       // Index 1
       IF "HMI_Interface_Overview".homeCodition[7].pageIndex = 1 THEN
           "HMI_Interface_Overview".homeCodition[7].emOverviewTitle := WSTRING#'Home Condition 1';
           "HMI_Interface_Overview".homeCodition[7].emOverviewCmName[0] := WSTRING#'Hot Press Right Servo Press';
           "HMI_Interface_Overview".homeCodition[7].emOverviewCmName[1] := WSTRING#'Hot Press Right Stage Lift Front';
           "HMI_Interface_Overview".homeCodition[7].emOverviewCmName[2] := WSTRING#'Hot Press Right Stage Lift Rear';
           "HMI_Interface_Overview".homeCodition[7].emOverviewCmName[3] := WSTRING#'Hot Press Right JR Detect';
           "HMI_Interface_Overview".homeCodition[7].emOverviewCmName[4] := WSTRING#'Spare';
           "HMI_Interface_Overview".homeCodition[7].emOverviewCmName[5] := WSTRING#'Spare';
           "HMI_Interface_Overview".homeCodition[7].emOverviewCmName[6] := WSTRING#'Spare';
           "HMI_Interface_Overview".homeCodition[7].emOverviewCmName[7] := WSTRING#'Spare';
           "HMI_Interface_Overview".homeCodition[7].emOverviewCmName[8] := WSTRING#'Spare';
           "HMI_Interface_Overview".homeCodition[7].emOverviewCmName[9] := WSTRING#'Spare';
           "HMI_Interface_Overview".homeCodition[7].emOverviewCmName[10] := WSTRING#'Spare';
           "HMI_Interface_Overview".homeCodition[7].emOverviewCmName[11] := WSTRING#'Spare';
           "HMI_Interface_Overview".homeCodition[7].emOverviewCmName[12] := WSTRING#'Spare';
           "HMI_Interface_Overview".homeCodition[7].emOverviewCmName[13] := WSTRING#'Spare';
           "HMI_Interface_Overview".homeCodition[7].emOverviewCmPositionName[0] := WSTRING#'Home Position';
           "HMI_Interface_Overview".homeCodition[7].emOverviewCmPositionName[1] := WSTRING#'Down';
           "HMI_Interface_Overview".homeCodition[7].emOverviewCmPositionName[2] := WSTRING#'Down';
           "HMI_Interface_Overview".homeCodition[7].emOverviewCmPositionName[3] := WSTRING#'Detect';
           "HMI_Interface_Overview".homeCodition[7].emOverviewCmPositionName[4] := WSTRING#'Spare';
           "HMI_Interface_Overview".homeCodition[7].emOverviewCmPositionName[5] := WSTRING#'Spare';
           "HMI_Interface_Overview".homeCodition[7].emOverviewCmPositionName[6] := WSTRING#'Spare';
           "HMI_Interface_Overview".homeCodition[7].emOverviewCmPositionName[7] := WSTRING#'Spare';
           "HMI_Interface_Overview".homeCodition[7].emOverviewCmPositionName[8] := WSTRING#'Spare';
           "HMI_Interface_Overview".homeCodition[7].emOverviewCmPositionName[9] := WSTRING#'Spare';
           "HMI_Interface_Overview".homeCodition[7].emOverviewCmPositionName[10] := WSTRING#'Spare';
           "HMI_Interface_Overview".homeCodition[7].emOverviewCmPositionName[11] := WSTRING#'Spare';
           "HMI_Interface_Overview".homeCodition[7].emOverviewCmPositionName[12] := WSTRING#'Spare';
           "HMI_Interface_Overview".homeCodition[7].emOverviewCmPositionName[13] := WSTRING#'Spare';
           IF NOT #statLampControl THEN
               "HMI_Interface_Overview".homeCodition[7].emOverviewHomeLampOn[0] := "Unit1.Em7.HmiInterface".cmHotPressRightServoPress.monitoring.profinetInput."HOME-POS-REACHED";
               "HMI_Interface_Overview".homeCodition[7].emOverviewHomeLampOn[1] := "Unit1.Em7.HmiInterface".cmHotPressRightStageLiftFrontUpDown.monitoring.inWorkPos;
               "HMI_Interface_Overview".homeCodition[7].emOverviewHomeLampOn[2] := "Unit1.Em7.HmiInterface".cmHotPressRightStageLiftRearUpDown.monitoring.inWorkPos;
               "HMI_Interface_Overview".homeCodition[7].emOverviewHomeLampOn[3] := "Unit1.Em7.HmiInterface".cmHotPressRightJRDetect.monitoring.processValue;
               "HMI_Interface_Overview".homeCodition[7].emOverviewHomeLampOn[4] := FALSE;
               "HMI_Interface_Overview".homeCodition[7].emOverviewHomeLampOn[5] := FALSE;
               "HMI_Interface_Overview".homeCodition[7].emOverviewHomeLampOn[6] := FALSE;
               "HMI_Interface_Overview".homeCodition[7].emOverviewHomeLampOn[7] := FALSE;
               "HMI_Interface_Overview".homeCodition[7].emOverviewHomeLampOn[8] := FALSE;
               "HMI_Interface_Overview".homeCodition[7].emOverviewHomeLampOn[9] := FALSE;
               "HMI_Interface_Overview".homeCodition[7].emOverviewHomeLampOn[10] := FALSE;
               "HMI_Interface_Overview".homeCodition[7].emOverviewHomeLampOn[11] := FALSE;
               "HMI_Interface_Overview".homeCodition[7].emOverviewHomeLampOn[12] := FALSE;
               "HMI_Interface_Overview".homeCodition[7].emOverviewHomeLampOn[13] := FALSE;
           END_IF;
       END_IF;

   END_REGION
END_REGION

REGION Network 38 (SCL): Em 8 Page Index Mapping
   REGION Page Index

       // Index 0
       IF "HMI_Interface_Overview".homeCodition[8].pageIndex = 0 THEN
           "HMI_Interface_Overview".homeCodition[8].emOverviewTitle := WSTRING#'Home Condition 0';
           "HMI_Interface_Overview".homeCodition[8].emOverviewCmName[0] := WSTRING#'Thickness Z-Axis';
           "HMI_Interface_Overview".homeCodition[8].emOverviewCmName[1] := WSTRING#'Hipot & Thickness Servo Press';
           "HMI_Interface_Overview".homeCodition[8].emOverviewCmName[2] := WSTRING#'Hipot Tab Contactor Left';
           "HMI_Interface_Overview".homeCodition[8].emOverviewCmName[3] := WSTRING#'Hipot Tab Contactor Right';
           "HMI_Interface_Overview".homeCodition[8].emOverviewCmName[4] := WSTRING#'Hipot Tab Contactor';
           "HMI_Interface_Overview".homeCodition[8].emOverviewCmName[5] := WSTRING#'Hipot & Thickness Stage Lift Front';
           "HMI_Interface_Overview".homeCodition[8].emOverviewCmName[6] := WSTRING#'Hipot & Thickness Stage Lift Rear';
           "HMI_Interface_Overview".homeCodition[8].emOverviewCmName[7] := WSTRING#'Hipot & Thickness JR Detect';
           "HMI_Interface_Overview".homeCodition[8].emOverviewCmName[8] := WSTRING#'Spare';
           "HMI_Interface_Overview".homeCodition[8].emOverviewCmName[9] := WSTRING#'Spare';
           "HMI_Interface_Overview".homeCodition[8].emOverviewCmName[10] := WSTRING#'Spare';
           "HMI_Interface_Overview".homeCodition[8].emOverviewCmName[11] := WSTRING#'Spare';
           "HMI_Interface_Overview".homeCodition[8].emOverviewCmName[12] := WSTRING#'Spare';
           "HMI_Interface_Overview".homeCodition[8].emOverviewCmName[13] := WSTRING#'Spare';
           "HMI_Interface_Overview".homeCodition[8].emOverviewCmPositionName[0] := WSTRING#'Wait Position';
           "HMI_Interface_Overview".homeCodition[8].emOverviewCmPositionName[1] := WSTRING#'Home Position';
           "HMI_Interface_Overview".homeCodition[8].emOverviewCmPositionName[2] := WSTRING#'Open';
           "HMI_Interface_Overview".homeCodition[8].emOverviewCmPositionName[3] := WSTRING#'Open';
           "HMI_Interface_Overview".homeCodition[8].emOverviewCmPositionName[4] := WSTRING#'Backward';
           "HMI_Interface_Overview".homeCodition[8].emOverviewCmPositionName[5] := WSTRING#'Down';
           "HMI_Interface_Overview".homeCodition[8].emOverviewCmPositionName[6] := WSTRING#'Down';
           "HMI_Interface_Overview".homeCodition[8].emOverviewCmPositionName[7] := WSTRING#'Not Detect';
           "HMI_Interface_Overview".homeCodition[8].emOverviewCmPositionName[8] := WSTRING#'Spare';
           "HMI_Interface_Overview".homeCodition[8].emOverviewCmPositionName[9] := WSTRING#'Spare';
           "HMI_Interface_Overview".homeCodition[8].emOverviewCmPositionName[10] := WSTRING#'Spare';
           "HMI_Interface_Overview".homeCodition[8].emOverviewCmPositionName[11] := WSTRING#'Spare';
           "HMI_Interface_Overview".homeCodition[8].emOverviewCmPositionName[12] := WSTRING#'Spare';
           "HMI_Interface_Overview".homeCodition[8].emOverviewCmPositionName[13] := WSTRING#'Spare';
           IF NOT #statLampControl THEN
               "HMI_Interface_Overview".homeCodition[8].emOverviewHomeLampOn[0] := "Unit1.Em8.HmiInterface".cm.softcam.thicknessAxisZ.pos00_wait.inPos;
               "HMI_Interface_Overview".homeCodition[8].emOverviewHomeLampOn[1] := "Unit1.Em8.HmiInterface".cmHipotThicknessServoPress.monitoring.profinetInput."HOME-POS-REACHED";
               "HMI_Interface_Overview".homeCodition[8].emOverviewHomeLampOn[2] := "Unit1.Em8.HmiInterface".cmHipotTabContactorLeftOpenClose.monitoring.inHomePos;
               "HMI_Interface_Overview".homeCodition[8].emOverviewHomeLampOn[3] := "Unit1.Em8.HmiInterface".cmHipotTabContactorRightOpenClose.monitoring.inHomePos;
               "HMI_Interface_Overview".homeCodition[8].emOverviewHomeLampOn[4] := "Unit1.Em8.HmiInterface".cmHipotTabContactorBwdFwd.monitoring.inHomePos;
               "HMI_Interface_Overview".homeCodition[8].emOverviewHomeLampOn[5] := "Unit1.Em8.HmiInterface".cmHipotThicknessStageLiftFrontUpDown.monitoring.inWorkPos;
               "HMI_Interface_Overview".homeCodition[8].emOverviewHomeLampOn[6] := "Unit1.Em8.HmiInterface".cmHipotThicknessStageLiftRearUpDown.monitoring.inWorkPos;
               "HMI_Interface_Overview".homeCodition[8].emOverviewHomeLampOn[7] := NOT "Unit1.Em8.HmiInterface".cmHipotThicknessJRDetect.monitoring.processValue;
               "HMI_Interface_Overview".homeCodition[8].emOverviewHomeLampOn[8] := FALSE;
               "HMI_Interface_Overview".homeCodition[8].emOverviewHomeLampOn[9] := FALSE;
               "HMI_Interface_Overview".homeCodition[8].emOverviewHomeLampOn[10] := FALSE;
               "HMI_Interface_Overview".homeCodition[8].emOverviewHomeLampOn[11] := FALSE;
               "HMI_Interface_Overview".homeCodition[8].emOverviewHomeLampOn[12] := FALSE;
               "HMI_Interface_Overview".homeCodition[8].emOverviewHomeLampOn[13] := FALSE;
           END_IF;
       END_IF;

       // Index 1
       IF "HMI_Interface_Overview".homeCodition[8].pageIndex = 1 THEN
           "HMI_Interface_Overview".homeCodition[8].emOverviewTitle := WSTRING#'Home Condition 1';
           "HMI_Interface_Overview".homeCodition[8].emOverviewCmName[0] := WSTRING#'Thickness Z-Axis';
           "HMI_Interface_Overview".homeCodition[8].emOverviewCmName[1] := WSTRING#'Hipot & Thickness Servo Press';
           "HMI_Interface_Overview".homeCodition[8].emOverviewCmName[2] := WSTRING#'Hipot Tab Contactor Left';
           "HMI_Interface_Overview".homeCodition[8].emOverviewCmName[3] := WSTRING#'Hipot Tab Contactor Right';
           "HMI_Interface_Overview".homeCodition[8].emOverviewCmName[4] := WSTRING#'Hipot Tab Contactor';
           "HMI_Interface_Overview".homeCodition[8].emOverviewCmName[5] := WSTRING#'Hipot & Thickness Stage Lift Front';
           "HMI_Interface_Overview".homeCodition[8].emOverviewCmName[6] := WSTRING#'Hipot & Thickness Stage Lift Rear';
           "HMI_Interface_Overview".homeCodition[8].emOverviewCmName[7] := WSTRING#'Hipot & Thickness JR Detect';
           "HMI_Interface_Overview".homeCodition[8].emOverviewCmName[8] := WSTRING#'Spare';
           "HMI_Interface_Overview".homeCodition[8].emOverviewCmName[9] := WSTRING#'Spare';
           "HMI_Interface_Overview".homeCodition[8].emOverviewCmName[10] := WSTRING#'Spare';
           "HMI_Interface_Overview".homeCodition[8].emOverviewCmName[11] := WSTRING#'Spare';
           "HMI_Interface_Overview".homeCodition[8].emOverviewCmName[12] := WSTRING#'Spare';
           "HMI_Interface_Overview".homeCodition[8].emOverviewCmName[13] := WSTRING#'Spare';
           "HMI_Interface_Overview".homeCodition[8].emOverviewCmPositionName[0] := WSTRING#'Wait Position';
           "HMI_Interface_Overview".homeCodition[8].emOverviewCmPositionName[1] := WSTRING#'Home Position';
           "HMI_Interface_Overview".homeCodition[8].emOverviewCmPositionName[2] := WSTRING#'Open';
           "HMI_Interface_Overview".homeCodition[8].emOverviewCmPositionName[3] := WSTRING#'Open';
           "HMI_Interface_Overview".homeCodition[8].emOverviewCmPositionName[4] := WSTRING#'Backward';
           "HMI_Interface_Overview".homeCodition[8].emOverviewCmPositionName[5] := WSTRING#'Down';
           "HMI_Interface_Overview".homeCodition[8].emOverviewCmPositionName[6] := WSTRING#'Down';
           "HMI_Interface_Overview".homeCodition[8].emOverviewCmPositionName[7] := WSTRING#'Detect';
           "HMI_Interface_Overview".homeCodition[8].emOverviewCmPositionName[8] := WSTRING#'Spare';
           "HMI_Interface_Overview".homeCodition[8].emOverviewCmPositionName[9] := WSTRING#'Spare';
           "HMI_Interface_Overview".homeCodition[8].emOverviewCmPositionName[10] := WSTRING#'Spare';
           "HMI_Interface_Overview".homeCodition[8].emOverviewCmPositionName[11] := WSTRING#'Spare';
           "HMI_Interface_Overview".homeCodition[8].emOverviewCmPositionName[12] := WSTRING#'Spare';
           "HMI_Interface_Overview".homeCodition[8].emOverviewCmPositionName[13] := WSTRING#'Spare';
           IF NOT #statLampControl THEN
               "HMI_Interface_Overview".homeCodition[8].emOverviewHomeLampOn[0] := "Unit1.Em8.HmiInterface".cm.softcam.thicknessAxisZ.pos00_wait.inPos;
               "HMI_Interface_Overview".homeCodition[8].emOverviewHomeLampOn[1] := "Unit1.Em8.HmiInterface".cmHipotThicknessServoPress.monitoring.profinetInput."HOME-POS-REACHED";
               "HMI_Interface_Overview".homeCodition[8].emOverviewHomeLampOn[2] := "Unit1.Em8.HmiInterface".cmHipotTabContactorLeftOpenClose.monitoring.inHomePos;
               "HMI_Interface_Overview".homeCodition[8].emOverviewHomeLampOn[3] := "Unit1.Em8.HmiInterface".cmHipotTabContactorRightOpenClose.monitoring.inHomePos;
               "HMI_Interface_Overview".homeCodition[8].emOverviewHomeLampOn[4] := "Unit1.Em8.HmiInterface".cmHipotTabContactorBwdFwd.monitoring.inHomePos;
               "HMI_Interface_Overview".homeCodition[8].emOverviewHomeLampOn[5] := "Unit1.Em8.HmiInterface".cmHipotThicknessStageLiftFrontUpDown.monitoring.inWorkPos;
               "HMI_Interface_Overview".homeCodition[8].emOverviewHomeLampOn[6] := "Unit1.Em8.HmiInterface".cmHipotThicknessStageLiftRearUpDown.monitoring.inWorkPos;
               "HMI_Interface_Overview".homeCodition[8].emOverviewHomeLampOn[7] := "Unit1.Em8.HmiInterface".cmHipotThicknessJRDetect.monitoring.processValue;
               "HMI_Interface_Overview".homeCodition[8].emOverviewHomeLampOn[8] := FALSE;
               "HMI_Interface_Overview".homeCodition[8].emOverviewHomeLampOn[9] := FALSE;
               "HMI_Interface_Overview".homeCodition[8].emOverviewHomeLampOn[10] := FALSE;
               "HMI_Interface_Overview".homeCodition[8].emOverviewHomeLampOn[11] := FALSE;
               "HMI_Interface_Overview".homeCodition[8].emOverviewHomeLampOn[12] := FALSE;
               "HMI_Interface_Overview".homeCodition[8].emOverviewHomeLampOn[13] := FALSE;
           END_IF;
       END_IF;

   END_REGION
END_REGION

REGION Network 39 (SCL): Em 9 Page Index Mapping
   REGION Page Index

       // Index 0
       IF "HMI_Interface_Overview".homeCodition[9].pageIndex = 0 THEN
           "HMI_Interface_Overview".homeCodition[9].emOverviewTitle := WSTRING#'Home Condition 0';
           "HMI_Interface_Overview".homeCodition[9].emOverviewCmName[0] := WSTRING#'Vision Stage Lift';
           "HMI_Interface_Overview".homeCodition[9].emOverviewCmName[1] := WSTRING#'Vision Light';
           "HMI_Interface_Overview".homeCodition[9].emOverviewCmName[2] := WSTRING#'Vision JR Detect';
           "HMI_Interface_Overview".homeCodition[9].emOverviewCmName[3] := WSTRING#'Spare';
           "HMI_Interface_Overview".homeCodition[9].emOverviewCmName[4] := WSTRING#'Spare';
           "HMI_Interface_Overview".homeCodition[9].emOverviewCmName[5] := WSTRING#'Spare';
           "HMI_Interface_Overview".homeCodition[9].emOverviewCmName[6] := WSTRING#'Spare';
           "HMI_Interface_Overview".homeCodition[9].emOverviewCmName[7] := WSTRING#'Spare';
           "HMI_Interface_Overview".homeCodition[9].emOverviewCmName[8] := WSTRING#'Spare';
           "HMI_Interface_Overview".homeCodition[9].emOverviewCmName[9] := WSTRING#'Spare';
           "HMI_Interface_Overview".homeCodition[9].emOverviewCmName[10] := WSTRING#'Spare';
           "HMI_Interface_Overview".homeCodition[9].emOverviewCmName[11] := WSTRING#'Spare';
           "HMI_Interface_Overview".homeCodition[9].emOverviewCmName[12] := WSTRING#'Spare';
           "HMI_Interface_Overview".homeCodition[9].emOverviewCmName[13] := WSTRING#'Spare';
           "HMI_Interface_Overview".homeCodition[9].emOverviewCmPositionName[0] := WSTRING#'Down';
           "HMI_Interface_Overview".homeCodition[9].emOverviewCmPositionName[1] := WSTRING#'Up';
           "HMI_Interface_Overview".homeCodition[9].emOverviewCmPositionName[2] := WSTRING#'Not Detect';
           "HMI_Interface_Overview".homeCodition[9].emOverviewCmPositionName[3] := WSTRING#'Spare';
           "HMI_Interface_Overview".homeCodition[9].emOverviewCmPositionName[4] := WSTRING#'Spare';
           "HMI_Interface_Overview".homeCodition[9].emOverviewCmPositionName[5] := WSTRING#'Spare';
           "HMI_Interface_Overview".homeCodition[9].emOverviewCmPositionName[6] := WSTRING#'Spare';
           "HMI_Interface_Overview".homeCodition[9].emOverviewCmPositionName[7] := WSTRING#'Spare';
           "HMI_Interface_Overview".homeCodition[9].emOverviewCmPositionName[8] := WSTRING#'Spare';
           "HMI_Interface_Overview".homeCodition[9].emOverviewCmPositionName[9] := WSTRING#'Spare';
           "HMI_Interface_Overview".homeCodition[9].emOverviewCmPositionName[10] := WSTRING#'Spare';
           "HMI_Interface_Overview".homeCodition[9].emOverviewCmPositionName[11] := WSTRING#'Spare';
           "HMI_Interface_Overview".homeCodition[9].emOverviewCmPositionName[12] := WSTRING#'Spare';
           "HMI_Interface_Overview".homeCodition[9].emOverviewCmPositionName[13] := WSTRING#'Spare';
           IF NOT #statLampControl THEN
               "HMI_Interface_Overview".homeCodition[9].emOverviewHomeLampOn[0] := "Unit1.Em9.HmiInterface".cmVisionStageLiftUpDown.monitoring.inWorkPos;
               "HMI_Interface_Overview".homeCodition[9].emOverviewHomeLampOn[1] := "Unit1.Em9.HmiInterface".cmVisionLightUpDown.monitoring.inHomePos;
               "HMI_Interface_Overview".homeCodition[9].emOverviewHomeLampOn[2] := NOT "Unit1.Em9.HmiInterface".cmVisionJRDetect.monitoring.processValue;
               "HMI_Interface_Overview".homeCodition[9].emOverviewHomeLampOn[3] := FALSE;
               "HMI_Interface_Overview".homeCodition[9].emOverviewHomeLampOn[4] := FALSE;
               "HMI_Interface_Overview".homeCodition[9].emOverviewHomeLampOn[5] := FALSE;
               "HMI_Interface_Overview".homeCodition[9].emOverviewHomeLampOn[6] := FALSE;
               "HMI_Interface_Overview".homeCodition[9].emOverviewHomeLampOn[7] := FALSE;
               "HMI_Interface_Overview".homeCodition[9].emOverviewHomeLampOn[8] := FALSE;
               "HMI_Interface_Overview".homeCodition[9].emOverviewHomeLampOn[9] := FALSE;
               "HMI_Interface_Overview".homeCodition[9].emOverviewHomeLampOn[10] := FALSE;
               "HMI_Interface_Overview".homeCodition[9].emOverviewHomeLampOn[11] := FALSE;
               "HMI_Interface_Overview".homeCodition[9].emOverviewHomeLampOn[12] := FALSE;
               "HMI_Interface_Overview".homeCodition[9].emOverviewHomeLampOn[13] := FALSE;
           END_IF;
       END_IF;

       // Index 1
       IF "HMI_Interface_Overview".homeCodition[9].pageIndex = 1 THEN
           "HMI_Interface_Overview".homeCodition[9].emOverviewTitle := WSTRING#'Home Condition 1';
           "HMI_Interface_Overview".homeCodition[9].emOverviewCmName[0] := WSTRING#'Vision Stage Lift';
           "HMI_Interface_Overview".homeCodition[9].emOverviewCmName[1] := WSTRING#'Vision Light';
           "HMI_Interface_Overview".homeCodition[9].emOverviewCmName[2] := WSTRING#'Vision JR Detect';
           "HMI_Interface_Overview".homeCodition[9].emOverviewCmName[3] := WSTRING#'Spare';
           "HMI_Interface_Overview".homeCodition[9].emOverviewCmName[4] := WSTRING#'Spare';
           "HMI_Interface_Overview".homeCodition[9].emOverviewCmName[5] := WSTRING#'Spare';
           "HMI_Interface_Overview".homeCodition[9].emOverviewCmName[6] := WSTRING#'Spare';
           "HMI_Interface_Overview".homeCodition[9].emOverviewCmName[7] := WSTRING#'Spare';
           "HMI_Interface_Overview".homeCodition[9].emOverviewCmName[8] := WSTRING#'Spare';
           "HMI_Interface_Overview".homeCodition[9].emOverviewCmName[9] := WSTRING#'Spare';
           "HMI_Interface_Overview".homeCodition[9].emOverviewCmName[10] := WSTRING#'Spare';
           "HMI_Interface_Overview".homeCodition[9].emOverviewCmName[11] := WSTRING#'Spare';
           "HMI_Interface_Overview".homeCodition[9].emOverviewCmName[12] := WSTRING#'Spare';
           "HMI_Interface_Overview".homeCodition[9].emOverviewCmName[13] := WSTRING#'Spare';
           "HMI_Interface_Overview".homeCodition[9].emOverviewCmPositionName[0] := WSTRING#'Down';
           "HMI_Interface_Overview".homeCodition[9].emOverviewCmPositionName[1] := WSTRING#'Up';
           "HMI_Interface_Overview".homeCodition[9].emOverviewCmPositionName[2] := WSTRING#'Detect';
           "HMI_Interface_Overview".homeCodition[9].emOverviewCmPositionName[3] := WSTRING#'Spare';
           "HMI_Interface_Overview".homeCodition[9].emOverviewCmPositionName[4] := WSTRING#'Spare';
           "HMI_Interface_Overview".homeCodition[9].emOverviewCmPositionName[5] := WSTRING#'Spare';
           "HMI_Interface_Overview".homeCodition[9].emOverviewCmPositionName[6] := WSTRING#'Spare';
           "HMI_Interface_Overview".homeCodition[9].emOverviewCmPositionName[7] := WSTRING#'Spare';
           "HMI_Interface_Overview".homeCodition[9].emOverviewCmPositionName[8] := WSTRING#'Spare';
           "HMI_Interface_Overview".homeCodition[9].emOverviewCmPositionName[9] := WSTRING#'Spare';
           "HMI_Interface_Overview".homeCodition[9].emOverviewCmPositionName[10] := WSTRING#'Spare';
           "HMI_Interface_Overview".homeCodition[9].emOverviewCmPositionName[11] := WSTRING#'Spare';
           "HMI_Interface_Overview".homeCodition[9].emOverviewCmPositionName[12] := WSTRING#'Spare';
           "HMI_Interface_Overview".homeCodition[9].emOverviewCmPositionName[13] := WSTRING#'Spare';
           IF NOT #statLampControl THEN
               "HMI_Interface_Overview".homeCodition[9].emOverviewHomeLampOn[0] := "Unit1.Em9.HmiInterface".cmVisionStageLiftUpDown.monitoring.inWorkPos;
               "HMI_Interface_Overview".homeCodition[9].emOverviewHomeLampOn[1] := "Unit1.Em9.HmiInterface".cmVisionLightUpDown.monitoring.inHomePos;
               "HMI_Interface_Overview".homeCodition[9].emOverviewHomeLampOn[2] := "Unit1.Em9.HmiInterface".cmVisionJRDetect.monitoring.processValue;
               "HMI_Interface_Overview".homeCodition[9].emOverviewHomeLampOn[3] := FALSE;
               "HMI_Interface_Overview".homeCodition[9].emOverviewHomeLampOn[4] := FALSE;
               "HMI_Interface_Overview".homeCodition[9].emOverviewHomeLampOn[5] := FALSE;
               "HMI_Interface_Overview".homeCodition[9].emOverviewHomeLampOn[6] := FALSE;
               "HMI_Interface_Overview".homeCodition[9].emOverviewHomeLampOn[7] := FALSE;
               "HMI_Interface_Overview".homeCodition[9].emOverviewHomeLampOn[8] := FALSE;
               "HMI_Interface_Overview".homeCodition[9].emOverviewHomeLampOn[9] := FALSE;
               "HMI_Interface_Overview".homeCodition[9].emOverviewHomeLampOn[10] := FALSE;
               "HMI_Interface_Overview".homeCodition[9].emOverviewHomeLampOn[11] := FALSE;
               "HMI_Interface_Overview".homeCodition[9].emOverviewHomeLampOn[12] := FALSE;
               "HMI_Interface_Overview".homeCodition[9].emOverviewHomeLampOn[13] := FALSE;
           END_IF;
       END_IF;

   END_REGION
END_REGION

REGION Network 40 (SCL): Em 10 Page Index Mapping
   REGION Page Index

       // Index 0
       IF "HMI_Interface_Overview".homeCodition[10].pageIndex = 0 THEN
           "HMI_Interface_Overview".homeCodition[10].emOverviewTitle := WSTRING#'Home Condition 0';
           "HMI_Interface_Overview".homeCodition[10].emOverviewCmName[0] := WSTRING#'Laser Mark Stage Lift';
           "HMI_Interface_Overview".homeCodition[10].emOverviewCmName[1] := WSTRING#'Laser Mark Cover';
           "HMI_Interface_Overview".homeCodition[10].emOverviewCmName[2] := WSTRING#'Laser Mark JR Detect';
           "HMI_Interface_Overview".homeCodition[10].emOverviewCmName[3] := WSTRING#'Spare';
           "HMI_Interface_Overview".homeCodition[10].emOverviewCmName[4] := WSTRING#'Spare';
           "HMI_Interface_Overview".homeCodition[10].emOverviewCmName[5] := WSTRING#'Spare';
           "HMI_Interface_Overview".homeCodition[10].emOverviewCmName[6] := WSTRING#'Spare';
           "HMI_Interface_Overview".homeCodition[10].emOverviewCmName[7] := WSTRING#'Spare';
           "HMI_Interface_Overview".homeCodition[10].emOverviewCmName[8] := WSTRING#'Spare';
           "HMI_Interface_Overview".homeCodition[10].emOverviewCmName[9] := WSTRING#'Spare';
           "HMI_Interface_Overview".homeCodition[10].emOverviewCmName[10] := WSTRING#'Spare';
           "HMI_Interface_Overview".homeCodition[10].emOverviewCmName[11] := WSTRING#'Spare';
           "HMI_Interface_Overview".homeCodition[10].emOverviewCmName[12] := WSTRING#'Spare';
           "HMI_Interface_Overview".homeCodition[10].emOverviewCmName[13] := WSTRING#'Spare';
           "HMI_Interface_Overview".homeCodition[10].emOverviewCmPositionName[0] := WSTRING#'Down';
           "HMI_Interface_Overview".homeCodition[10].emOverviewCmPositionName[1] := WSTRING#'Up';
           "HMI_Interface_Overview".homeCodition[10].emOverviewCmPositionName[2] := WSTRING#'Not Detect';
           "HMI_Interface_Overview".homeCodition[10].emOverviewCmPositionName[3] := WSTRING#'Spare';
           "HMI_Interface_Overview".homeCodition[10].emOverviewCmPositionName[4] := WSTRING#'Spare';
           "HMI_Interface_Overview".homeCodition[10].emOverviewCmPositionName[5] := WSTRING#'Spare';
           "HMI_Interface_Overview".homeCodition[10].emOverviewCmPositionName[6] := WSTRING#'Spare';
           "HMI_Interface_Overview".homeCodition[10].emOverviewCmPositionName[7] := WSTRING#'Spare';
           "HMI_Interface_Overview".homeCodition[10].emOverviewCmPositionName[8] := WSTRING#'Spare';
           "HMI_Interface_Overview".homeCodition[10].emOverviewCmPositionName[9] := WSTRING#'Spare';
           "HMI_Interface_Overview".homeCodition[10].emOverviewCmPositionName[10] := WSTRING#'Spare';
           "HMI_Interface_Overview".homeCodition[10].emOverviewCmPositionName[11] := WSTRING#'Spare';
           "HMI_Interface_Overview".homeCodition[10].emOverviewCmPositionName[12] := WSTRING#'Spare';
           "HMI_Interface_Overview".homeCodition[10].emOverviewCmPositionName[13] := WSTRING#'Spare';
           IF NOT #statLampControl THEN
               "HMI_Interface_Overview".homeCodition[10].emOverviewHomeLampOn[0] := "Unit1.Em10.HmiInterface".cmLaserMarkStageLiftUpDown.monitoring.inWorkPos;
               "HMI_Interface_Overview".homeCodition[10].emOverviewHomeLampOn[1] := "Unit1.Em10.HmiInterface".cmLaserMarkCoverUpDown.monitoring.inHomePos;
               "HMI_Interface_Overview".homeCodition[10].emOverviewHomeLampOn[2] := NOT "Unit1.Em10.HmiInterface".cmLaserMarkJRDetect.monitoring.processValue;
               "HMI_Interface_Overview".homeCodition[10].emOverviewHomeLampOn[3] := FALSE;
               "HMI_Interface_Overview".homeCodition[10].emOverviewHomeLampOn[4] := FALSE;
               "HMI_Interface_Overview".homeCodition[10].emOverviewHomeLampOn[5] := FALSE;
               "HMI_Interface_Overview".homeCodition[10].emOverviewHomeLampOn[6] := FALSE;
               "HMI_Interface_Overview".homeCodition[10].emOverviewHomeLampOn[7] := FALSE;
               "HMI_Interface_Overview".homeCodition[10].emOverviewHomeLampOn[8] := FALSE;
               "HMI_Interface_Overview".homeCodition[10].emOverviewHomeLampOn[9] := FALSE;
               "HMI_Interface_Overview".homeCodition[10].emOverviewHomeLampOn[10] := FALSE;
               "HMI_Interface_Overview".homeCodition[10].emOverviewHomeLampOn[11] := FALSE;
               "HMI_Interface_Overview".homeCodition[10].emOverviewHomeLampOn[12] := FALSE;
               "HMI_Interface_Overview".homeCodition[10].emOverviewHomeLampOn[13] := FALSE;
           END_IF;
       END_IF;

       // Index 1
       IF "HMI_Interface_Overview".homeCodition[10].pageIndex = 1 THEN
           "HMI_Interface_Overview".homeCodition[10].emOverviewTitle := WSTRING#'Home Condition 1';
           "HMI_Interface_Overview".homeCodition[10].emOverviewCmName[0] := WSTRING#'Laser Mark Stage Lift';
           "HMI_Interface_Overview".homeCodition[10].emOverviewCmName[1] := WSTRING#'Laser Mark Cover';
           "HMI_Interface_Overview".homeCodition[10].emOverviewCmName[2] := WSTRING#'Laser Mark JR Detect';
           "HMI_Interface_Overview".homeCodition[10].emOverviewCmName[3] := WSTRING#'Spare';
           "HMI_Interface_Overview".homeCodition[10].emOverviewCmName[4] := WSTRING#'Spare';
           "HMI_Interface_Overview".homeCodition[10].emOverviewCmName[5] := WSTRING#'Spare';
           "HMI_Interface_Overview".homeCodition[10].emOverviewCmName[6] := WSTRING#'Spare';
           "HMI_Interface_Overview".homeCodition[10].emOverviewCmName[7] := WSTRING#'Spare';
           "HMI_Interface_Overview".homeCodition[10].emOverviewCmName[8] := WSTRING#'Spare';
           "HMI_Interface_Overview".homeCodition[10].emOverviewCmName[9] := WSTRING#'Spare';
           "HMI_Interface_Overview".homeCodition[10].emOverviewCmName[10] := WSTRING#'Spare';
           "HMI_Interface_Overview".homeCodition[10].emOverviewCmName[11] := WSTRING#'Spare';
           "HMI_Interface_Overview".homeCodition[10].emOverviewCmName[12] := WSTRING#'Spare';
           "HMI_Interface_Overview".homeCodition[10].emOverviewCmName[13] := WSTRING#'Spare';
           "HMI_Interface_Overview".homeCodition[10].emOverviewCmPositionName[0] := WSTRING#'Down';
           "HMI_Interface_Overview".homeCodition[10].emOverviewCmPositionName[1] := WSTRING#'Up';
           "HMI_Interface_Overview".homeCodition[10].emOverviewCmPositionName[2] := WSTRING#'Detect';
           "HMI_Interface_Overview".homeCodition[10].emOverviewCmPositionName[3] := WSTRING#'Spare';
           "HMI_Interface_Overview".homeCodition[10].emOverviewCmPositionName[4] := WSTRING#'Spare';
           "HMI_Interface_Overview".homeCodition[10].emOverviewCmPositionName[5] := WSTRING#'Spare';
           "HMI_Interface_Overview".homeCodition[10].emOverviewCmPositionName[6] := WSTRING#'Spare';
           "HMI_Interface_Overview".homeCodition[10].emOverviewCmPositionName[7] := WSTRING#'Spare';
           "HMI_Interface_Overview".homeCodition[10].emOverviewCmPositionName[8] := WSTRING#'Spare';
           "HMI_Interface_Overview".homeCodition[10].emOverviewCmPositionName[9] := WSTRING#'Spare';
           "HMI_Interface_Overview".homeCodition[10].emOverviewCmPositionName[10] := WSTRING#'Spare';
           "HMI_Interface_Overview".homeCodition[10].emOverviewCmPositionName[11] := WSTRING#'Spare';
           "HMI_Interface_Overview".homeCodition[10].emOverviewCmPositionName[12] := WSTRING#'Spare';
           "HMI_Interface_Overview".homeCodition[10].emOverviewCmPositionName[13] := WSTRING#'Spare';
           IF NOT #statLampControl THEN
               "HMI_Interface_Overview".homeCodition[10].emOverviewHomeLampOn[0] := "Unit1.Em10.HmiInterface".cmLaserMarkStageLiftUpDown.monitoring.inWorkPos;
               "HMI_Interface_Overview".homeCodition[10].emOverviewHomeLampOn[1] := "Unit1.Em10.HmiInterface".cmLaserMarkCoverUpDown.monitoring.inHomePos;
               "HMI_Interface_Overview".homeCodition[10].emOverviewHomeLampOn[2] := "Unit1.Em10.HmiInterface".cmLaserMarkJRDetect.monitoring.processValue;
               "HMI_Interface_Overview".homeCodition[10].emOverviewHomeLampOn[3] := FALSE;
               "HMI_Interface_Overview".homeCodition[10].emOverviewHomeLampOn[4] := FALSE;
               "HMI_Interface_Overview".homeCodition[10].emOverviewHomeLampOn[5] := FALSE;
               "HMI_Interface_Overview".homeCodition[10].emOverviewHomeLampOn[6] := FALSE;
               "HMI_Interface_Overview".homeCodition[10].emOverviewHomeLampOn[7] := FALSE;
               "HMI_Interface_Overview".homeCodition[10].emOverviewHomeLampOn[8] := FALSE;
               "HMI_Interface_Overview".homeCodition[10].emOverviewHomeLampOn[9] := FALSE;
               "HMI_Interface_Overview".homeCodition[10].emOverviewHomeLampOn[10] := FALSE;
               "HMI_Interface_Overview".homeCodition[10].emOverviewHomeLampOn[11] := FALSE;
               "HMI_Interface_Overview".homeCodition[10].emOverviewHomeLampOn[12] := FALSE;
               "HMI_Interface_Overview".homeCodition[10].emOverviewHomeLampOn[13] := FALSE;
           END_IF;
       END_IF;

   END_REGION
END_REGION

REGION Network 41 (SCL): Em 12 Page Index Mapping
   REGION Page Index

       // Index 0
       IF "HMI_Interface_Overview".homeCodition[12].pageIndex = 0 THEN
           "HMI_Interface_Overview".homeCodition[12].emOverviewTitle := WSTRING#'Home Condition 0';
           "HMI_Interface_Overview".homeCodition[12].emOverviewCmName[0] := WSTRING#'Stack NG Box Loading';
           "HMI_Interface_Overview".homeCodition[12].emOverviewCmName[1] := WSTRING#'Stack NG Box Unit Mover';
           "HMI_Interface_Overview".homeCodition[12].emOverviewCmName[2] := WSTRING#'Stack NG Box Clamp Left ';
           "HMI_Interface_Overview".homeCodition[12].emOverviewCmName[3] := WSTRING#'Stack NG Box Clamp Right';
           "HMI_Interface_Overview".homeCodition[12].emOverviewCmName[4] := WSTRING#'Stack NG Box Clamp Mover';
           "HMI_Interface_Overview".homeCodition[12].emOverviewCmName[5] := WSTRING#'Spare';
           "HMI_Interface_Overview".homeCodition[12].emOverviewCmName[6] := WSTRING#'Spare';
           "HMI_Interface_Overview".homeCodition[12].emOverviewCmName[7] := WSTRING#'Spare';
           "HMI_Interface_Overview".homeCodition[12].emOverviewCmName[8] := WSTRING#'Spare';
           "HMI_Interface_Overview".homeCodition[12].emOverviewCmName[9] := WSTRING#'Spare';
           "HMI_Interface_Overview".homeCodition[12].emOverviewCmName[10] := WSTRING#'Spare';
           "HMI_Interface_Overview".homeCodition[12].emOverviewCmName[11] := WSTRING#'Spare';
           "HMI_Interface_Overview".homeCodition[12].emOverviewCmName[12] := WSTRING#'Spare';
           "HMI_Interface_Overview".homeCodition[12].emOverviewCmName[13] := WSTRING#'Spare';
           "HMI_Interface_Overview".homeCodition[12].emOverviewCmPositionName[0] := WSTRING#'Up';
           "HMI_Interface_Overview".homeCodition[12].emOverviewCmPositionName[1] := WSTRING#'Forward';
           "HMI_Interface_Overview".homeCodition[12].emOverviewCmPositionName[2] := WSTRING#'Open';
           "HMI_Interface_Overview".homeCodition[12].emOverviewCmPositionName[3] := WSTRING#'Open';
           "HMI_Interface_Overview".homeCodition[12].emOverviewCmPositionName[4] := WSTRING#'Open';
           "HMI_Interface_Overview".homeCodition[12].emOverviewCmPositionName[5] := WSTRING#'Spare';
           "HMI_Interface_Overview".homeCodition[12].emOverviewCmPositionName[6] := WSTRING#'Spare';
           "HMI_Interface_Overview".homeCodition[12].emOverviewCmPositionName[7] := WSTRING#'Spare';
           "HMI_Interface_Overview".homeCodition[12].emOverviewCmPositionName[8] := WSTRING#'Spare';
           "HMI_Interface_Overview".homeCodition[12].emOverviewCmPositionName[9] := WSTRING#'Spare';
           "HMI_Interface_Overview".homeCodition[12].emOverviewCmPositionName[10] := WSTRING#'Spare';
           "HMI_Interface_Overview".homeCodition[12].emOverviewCmPositionName[11] := WSTRING#'Spare';
           "HMI_Interface_Overview".homeCodition[12].emOverviewCmPositionName[12] := WSTRING#'Spare';
           "HMI_Interface_Overview".homeCodition[12].emOverviewCmPositionName[13] := WSTRING#'Spare';
           IF NOT #statLampControl THEN
               "HMI_Interface_Overview".homeCodition[12].emOverviewHomeLampOn[0] := "Unit1.Em12.HmiInterface".cmStackNgBoxLoadingUpDown.monitoring.inHomePos;
               "HMI_Interface_Overview".homeCodition[12].emOverviewHomeLampOn[1] := "Unit1.Em12.HmiInterface".cmStackNgBoxUnitMoverBwdFwd.monitoring.inWorkPos;
               "HMI_Interface_Overview".homeCodition[12].emOverviewHomeLampOn[2] := "Unit1.Em12.HmiInterface".cmStackNgBoxClampLeftOpenClose.monitoring.inHomePos;
               "HMI_Interface_Overview".homeCodition[12].emOverviewHomeLampOn[3] := "Unit1.Em12.HmiInterface".cmStackNgBoxClampRightOpenClose.monitoring.inHomePos;
               "HMI_Interface_Overview".homeCodition[12].emOverviewHomeLampOn[4] := "Unit1.Em12.HmiInterface".cmStackNgBoxClampMoverOpenClose.monitoring.inHomePos;
               "HMI_Interface_Overview".homeCodition[12].emOverviewHomeLampOn[5] := FALSE;
               "HMI_Interface_Overview".homeCodition[12].emOverviewHomeLampOn[6] := FALSE;
               "HMI_Interface_Overview".homeCodition[12].emOverviewHomeLampOn[7] := FALSE;
               "HMI_Interface_Overview".homeCodition[12].emOverviewHomeLampOn[8] := FALSE;
               "HMI_Interface_Overview".homeCodition[12].emOverviewHomeLampOn[9] := FALSE;
               "HMI_Interface_Overview".homeCodition[12].emOverviewHomeLampOn[10] := FALSE;
               "HMI_Interface_Overview".homeCodition[12].emOverviewHomeLampOn[11] := FALSE;
               "HMI_Interface_Overview".homeCodition[12].emOverviewHomeLampOn[12] := FALSE;
               "HMI_Interface_Overview".homeCodition[12].emOverviewHomeLampOn[13] := FALSE;
           END_IF;
       END_IF;

       // Index 1
       IF "HMI_Interface_Overview".homeCodition[12].pageIndex = 1 THEN
           "HMI_Interface_Overview".homeCodition[12].emOverviewTitle := WSTRING#'Home Condition 1';
           "HMI_Interface_Overview".homeCodition[12].emOverviewCmName[0] := WSTRING#'Stack NG Box Loading';
           "HMI_Interface_Overview".homeCodition[12].emOverviewCmName[1] := WSTRING#'Stack NG Box Unit Mover';
           "HMI_Interface_Overview".homeCodition[12].emOverviewCmName[2] := WSTRING#'Stack NG Box Clamp Left ';
           "HMI_Interface_Overview".homeCodition[12].emOverviewCmName[3] := WSTRING#'Stack NG Box Clamp Right';
           "HMI_Interface_Overview".homeCodition[12].emOverviewCmName[4] := WSTRING#'Stack NG Box Clamp Mover';
           "HMI_Interface_Overview".homeCodition[12].emOverviewCmName[5] := WSTRING#'Spare';
           "HMI_Interface_Overview".homeCodition[12].emOverviewCmName[6] := WSTRING#'Spare';
           "HMI_Interface_Overview".homeCodition[12].emOverviewCmName[7] := WSTRING#'Spare';
           "HMI_Interface_Overview".homeCodition[12].emOverviewCmName[8] := WSTRING#'Spare';
           "HMI_Interface_Overview".homeCodition[12].emOverviewCmName[9] := WSTRING#'Spare';
           "HMI_Interface_Overview".homeCodition[12].emOverviewCmName[10] := WSTRING#'Spare';
           "HMI_Interface_Overview".homeCodition[12].emOverviewCmName[11] := WSTRING#'Spare';
           "HMI_Interface_Overview".homeCodition[12].emOverviewCmName[12] := WSTRING#'Spare';
           "HMI_Interface_Overview".homeCodition[12].emOverviewCmName[13] := WSTRING#'Spare';
           "HMI_Interface_Overview".homeCodition[12].emOverviewCmPositionName[0] := WSTRING#'Up';
           "HMI_Interface_Overview".homeCodition[12].emOverviewCmPositionName[1] := WSTRING#'Forward';
           "HMI_Interface_Overview".homeCodition[12].emOverviewCmPositionName[2] := WSTRING#'Close';
           "HMI_Interface_Overview".homeCodition[12].emOverviewCmPositionName[3] := WSTRING#'Close';
           "HMI_Interface_Overview".homeCodition[12].emOverviewCmPositionName[4] := WSTRING#'Close';
           "HMI_Interface_Overview".homeCodition[12].emOverviewCmPositionName[5] := WSTRING#'Spare';
           "HMI_Interface_Overview".homeCodition[12].emOverviewCmPositionName[6] := WSTRING#'Spare';
           "HMI_Interface_Overview".homeCodition[12].emOverviewCmPositionName[7] := WSTRING#'Spare';
           "HMI_Interface_Overview".homeCodition[12].emOverviewCmPositionName[8] := WSTRING#'Spare';
           "HMI_Interface_Overview".homeCodition[12].emOverviewCmPositionName[9] := WSTRING#'Spare';
           "HMI_Interface_Overview".homeCodition[12].emOverviewCmPositionName[10] := WSTRING#'Spare';
           "HMI_Interface_Overview".homeCodition[12].emOverviewCmPositionName[11] := WSTRING#'Spare';
           "HMI_Interface_Overview".homeCodition[12].emOverviewCmPositionName[12] := WSTRING#'Spare';
           "HMI_Interface_Overview".homeCodition[12].emOverviewCmPositionName[13] := WSTRING#'Spare';
           IF NOT #statLampControl THEN
               "HMI_Interface_Overview".homeCodition[12].emOverviewHomeLampOn[0] := "Unit1.Em12.HmiInterface".cmStackNgBoxLoadingUpDown.monitoring.inHomePos;
               "HMI_Interface_Overview".homeCodition[12].emOverviewHomeLampOn[1] := "Unit1.Em12.HmiInterface".cmStackNgBoxUnitMoverBwdFwd.monitoring.inWorkPos;
               "HMI_Interface_Overview".homeCodition[12].emOverviewHomeLampOn[2] := "Unit1.Em12.HmiInterface".cmStackNgBoxClampLeftOpenClose.monitoring.inWorkPos;
               "HMI_Interface_Overview".homeCodition[12].emOverviewHomeLampOn[3] := "Unit1.Em12.HmiInterface".cmStackNgBoxClampRightOpenClose.monitoring.inWorkPos;
               "HMI_Interface_Overview".homeCodition[12].emOverviewHomeLampOn[4] := "Unit1.Em12.HmiInterface".cmStackNgBoxClampMoverOpenClose.monitoring.inWorkPos;
               "HMI_Interface_Overview".homeCodition[12].emOverviewHomeLampOn[5] := FALSE;
               "HMI_Interface_Overview".homeCodition[12].emOverviewHomeLampOn[6] := FALSE;
               "HMI_Interface_Overview".homeCodition[12].emOverviewHomeLampOn[7] := FALSE;
               "HMI_Interface_Overview".homeCodition[12].emOverviewHomeLampOn[8] := FALSE;
               "HMI_Interface_Overview".homeCodition[12].emOverviewHomeLampOn[9] := FALSE;
               "HMI_Interface_Overview".homeCodition[12].emOverviewHomeLampOn[10] := FALSE;
               "HMI_Interface_Overview".homeCodition[12].emOverviewHomeLampOn[11] := FALSE;
               "HMI_Interface_Overview".homeCodition[12].emOverviewHomeLampOn[12] := FALSE;
               "HMI_Interface_Overview".homeCodition[12].emOverviewHomeLampOn[13] := FALSE;
           END_IF;
       END_IF;

   END_REGION
END_REGION

REGION Network 42 (SCL): Em 13 Page Index Mapping
   REGION Page Index

       // Index 0
       IF "HMI_Interface_Overview".homeCodition[13].pageIndex = 0 THEN
           "HMI_Interface_Overview".homeCodition[13].emOverviewTitle := WSTRING#'Home Condition 0';
           "HMI_Interface_Overview".homeCodition[13].emOverviewCmName[0] := WSTRING#'JR Unloading P&P X-Axis';
           "HMI_Interface_Overview".homeCodition[13].emOverviewCmName[1] := WSTRING#'JR Unloading P&P Z-Axis';
           "HMI_Interface_Overview".homeCodition[13].emOverviewCmName[2] := WSTRING#'JR Unloading P&P C-Axis';
           "HMI_Interface_Overview".homeCodition[13].emOverviewCmName[3] := WSTRING#'JR Unloading P&P Clamp';
           "HMI_Interface_Overview".homeCodition[13].emOverviewCmName[4] := WSTRING#'JR Unloading P&P JR Detect';
           "HMI_Interface_Overview".homeCodition[13].emOverviewCmName[5] := WSTRING#'Spare';
           "HMI_Interface_Overview".homeCodition[13].emOverviewCmName[6] := WSTRING#'Spare';
           "HMI_Interface_Overview".homeCodition[13].emOverviewCmName[7] := WSTRING#'Spare';
           "HMI_Interface_Overview".homeCodition[13].emOverviewCmName[8] := WSTRING#'Spare';
           "HMI_Interface_Overview".homeCodition[13].emOverviewCmName[9] := WSTRING#'Spare';
           "HMI_Interface_Overview".homeCodition[13].emOverviewCmName[10] := WSTRING#'Spare';
           "HMI_Interface_Overview".homeCodition[13].emOverviewCmName[11] := WSTRING#'Spare';
           "HMI_Interface_Overview".homeCodition[13].emOverviewCmName[12] := WSTRING#'Spare';
           "HMI_Interface_Overview".homeCodition[13].emOverviewCmName[13] := WSTRING#'Spare';
           "HMI_Interface_Overview".homeCodition[13].emOverviewCmPositionName[0] := WSTRING#'Wait Position';
           "HMI_Interface_Overview".homeCodition[13].emOverviewCmPositionName[1] := WSTRING#'Wait Position';
           "HMI_Interface_Overview".homeCodition[13].emOverviewCmPositionName[2] := WSTRING#'Wait Position';
           "HMI_Interface_Overview".homeCodition[13].emOverviewCmPositionName[3] := WSTRING#'Open';
           "HMI_Interface_Overview".homeCodition[13].emOverviewCmPositionName[4] := WSTRING#'Not Detect';
           "HMI_Interface_Overview".homeCodition[13].emOverviewCmPositionName[5] := WSTRING#'Spare';
           "HMI_Interface_Overview".homeCodition[13].emOverviewCmPositionName[6] := WSTRING#'Spare';
           "HMI_Interface_Overview".homeCodition[13].emOverviewCmPositionName[7] := WSTRING#'Spare';
           "HMI_Interface_Overview".homeCodition[13].emOverviewCmPositionName[8] := WSTRING#'Spare';
           "HMI_Interface_Overview".homeCodition[13].emOverviewCmPositionName[9] := WSTRING#'Spare';
           "HMI_Interface_Overview".homeCodition[13].emOverviewCmPositionName[10] := WSTRING#'Spare';
           "HMI_Interface_Overview".homeCodition[13].emOverviewCmPositionName[11] := WSTRING#'Spare';
           "HMI_Interface_Overview".homeCodition[13].emOverviewCmPositionName[12] := WSTRING#'Spare';
           "HMI_Interface_Overview".homeCodition[13].emOverviewCmPositionName[13] := WSTRING#'Spare';
           IF NOT #statLampControl THEN
               "HMI_Interface_Overview".homeCodition[13].emOverviewHomeLampOn[0] := "Unit1.Em13.HmiInterface".cm.softcam.jrUnIoadingPnPAxisX.pos00_wait.inPos;
               "HMI_Interface_Overview".homeCodition[13].emOverviewHomeLampOn[1] := "Unit1.Em13.HmiInterface".cm.softcam.jrUnIoadingPnPAxisZ.pos00_wait.inPos;
               "HMI_Interface_Overview".homeCodition[13].emOverviewHomeLampOn[2] := "Unit1.Em13.HmiInterface".cm.softcam.jrUnIoadingPnPAxisC.pos00_wait.inPos;
               "HMI_Interface_Overview".homeCodition[13].emOverviewHomeLampOn[3] := "Unit1.Em13.HmiInterface".cmJRUnloadingPnPClampOpenClose.monitoring.inHomePos;
               "HMI_Interface_Overview".homeCodition[13].emOverviewHomeLampOn[4] := NOT "Unit1.Em13.HmiInterface".cmJRUnloadingPnPJRDetect.monitoring.processValue;
               "HMI_Interface_Overview".homeCodition[13].emOverviewHomeLampOn[5] := FALSE;
               "HMI_Interface_Overview".homeCodition[13].emOverviewHomeLampOn[6] := FALSE;
               "HMI_Interface_Overview".homeCodition[13].emOverviewHomeLampOn[7] := FALSE;
               "HMI_Interface_Overview".homeCodition[13].emOverviewHomeLampOn[8] := FALSE;
               "HMI_Interface_Overview".homeCodition[13].emOverviewHomeLampOn[9] := FALSE;
               "HMI_Interface_Overview".homeCodition[13].emOverviewHomeLampOn[10] := FALSE;
               "HMI_Interface_Overview".homeCodition[13].emOverviewHomeLampOn[11] := FALSE;
               "HMI_Interface_Overview".homeCodition[13].emOverviewHomeLampOn[12] := FALSE;
               "HMI_Interface_Overview".homeCodition[13].emOverviewHomeLampOn[13] := FALSE;
           END_IF;
       END_IF;

       // Index 1
       IF "HMI_Interface_Overview".homeCodition[13].pageIndex = 1 THEN
           "HMI_Interface_Overview".homeCodition[13].emOverviewTitle := WSTRING#'Home Condition 1';
           "HMI_Interface_Overview".homeCodition[13].emOverviewCmName[0] := WSTRING#'JR Unloading P&P X-Axis';
           "HMI_Interface_Overview".homeCodition[13].emOverviewCmName[1] := WSTRING#'JR Unloading P&P Z-Axis';
           "HMI_Interface_Overview".homeCodition[13].emOverviewCmName[2] := WSTRING#'JR Unloading P&P C-Axis';
           "HMI_Interface_Overview".homeCodition[13].emOverviewCmName[3] := WSTRING#'JR Unloading P&P Clamp';
           "HMI_Interface_Overview".homeCodition[13].emOverviewCmName[4] := WSTRING#'JR Unloading P&P JR Detect';
           "HMI_Interface_Overview".homeCodition[13].emOverviewCmName[5] := WSTRING#'Spare';
           "HMI_Interface_Overview".homeCodition[13].emOverviewCmName[6] := WSTRING#'Spare';
           "HMI_Interface_Overview".homeCodition[13].emOverviewCmName[7] := WSTRING#'Spare';
           "HMI_Interface_Overview".homeCodition[13].emOverviewCmName[8] := WSTRING#'Spare';
           "HMI_Interface_Overview".homeCodition[13].emOverviewCmName[9] := WSTRING#'Spare';
           "HMI_Interface_Overview".homeCodition[13].emOverviewCmName[10] := WSTRING#'Spare';
           "HMI_Interface_Overview".homeCodition[13].emOverviewCmName[11] := WSTRING#'Spare';
           "HMI_Interface_Overview".homeCodition[13].emOverviewCmName[12] := WSTRING#'Spare';
           "HMI_Interface_Overview".homeCodition[13].emOverviewCmName[13] := WSTRING#'Spare';
           "HMI_Interface_Overview".homeCodition[13].emOverviewCmPositionName[0] := WSTRING#'Wait Position';
           "HMI_Interface_Overview".homeCodition[13].emOverviewCmPositionName[1] := WSTRING#'Wait Position';
           "HMI_Interface_Overview".homeCodition[13].emOverviewCmPositionName[2] := WSTRING#'Wait Position';
           "HMI_Interface_Overview".homeCodition[13].emOverviewCmPositionName[3] := WSTRING#'Close';
           "HMI_Interface_Overview".homeCodition[13].emOverviewCmPositionName[4] := WSTRING#'Detect';
           "HMI_Interface_Overview".homeCodition[13].emOverviewCmPositionName[5] := WSTRING#'Spare';
           "HMI_Interface_Overview".homeCodition[13].emOverviewCmPositionName[6] := WSTRING#'Spare';
           "HMI_Interface_Overview".homeCodition[13].emOverviewCmPositionName[7] := WSTRING#'Spare';
           "HMI_Interface_Overview".homeCodition[13].emOverviewCmPositionName[8] := WSTRING#'Spare';
           "HMI_Interface_Overview".homeCodition[13].emOverviewCmPositionName[9] := WSTRING#'Spare';
           "HMI_Interface_Overview".homeCodition[13].emOverviewCmPositionName[10] := WSTRING#'Spare';
           "HMI_Interface_Overview".homeCodition[13].emOverviewCmPositionName[11] := WSTRING#'Spare';
           "HMI_Interface_Overview".homeCodition[13].emOverviewCmPositionName[12] := WSTRING#'Spare';
           "HMI_Interface_Overview".homeCodition[13].emOverviewCmPositionName[13] := WSTRING#'Spare';
           IF NOT #statLampControl THEN
               "HMI_Interface_Overview".homeCodition[13].emOverviewHomeLampOn[0] := "Unit1.Em13.HmiInterface".cm.softcam.jrUnIoadingPnPAxisX.pos00_wait.inPos;
               "HMI_Interface_Overview".homeCodition[13].emOverviewHomeLampOn[1] := "Unit1.Em13.HmiInterface".cm.softcam.jrUnIoadingPnPAxisZ.pos00_wait.inPos;
               "HMI_Interface_Overview".homeCodition[13].emOverviewHomeLampOn[2] := "Unit1.Em13.HmiInterface".cm.softcam.jrUnIoadingPnPAxisC.pos00_wait.inPos;
               "HMI_Interface_Overview".homeCodition[13].emOverviewHomeLampOn[3] := "Unit1.Em13.HmiInterface".cmJRUnloadingPnPClampOpenClose.monitoring.inWorkPos;
               "HMI_Interface_Overview".homeCodition[13].emOverviewHomeLampOn[4] := "Unit1.Em13.HmiInterface".cmJRUnloadingPnPJRDetect.monitoring.processValue;
               "HMI_Interface_Overview".homeCodition[13].emOverviewHomeLampOn[5] := FALSE;
               "HMI_Interface_Overview".homeCodition[13].emOverviewHomeLampOn[6] := FALSE;
               "HMI_Interface_Overview".homeCodition[13].emOverviewHomeLampOn[7] := FALSE;
               "HMI_Interface_Overview".homeCodition[13].emOverviewHomeLampOn[8] := FALSE;
               "HMI_Interface_Overview".homeCodition[13].emOverviewHomeLampOn[9] := FALSE;
               "HMI_Interface_Overview".homeCodition[13].emOverviewHomeLampOn[10] := FALSE;
               "HMI_Interface_Overview".homeCodition[13].emOverviewHomeLampOn[11] := FALSE;
               "HMI_Interface_Overview".homeCodition[13].emOverviewHomeLampOn[12] := FALSE;
               "HMI_Interface_Overview".homeCodition[13].emOverviewHomeLampOn[13] := FALSE;
           END_IF;
       END_IF;

   END_REGION
END_REGION
END_FUNCTION_BLOCK
